Staubli VAL3: sendCommand.pgx

program sendCommand(num x_nCamID (dimensions=1), string x_sCmd (dimensions=1), bool& x_bError[] (dimensions=1))
  local string l_sMsgError
  local bool l_bError
  local num l_nErrorCode
begin
  //-----------------------------------------------------------------------
  //Header begin
  //Description of program
  //  Send native command to camera and read command execution error.
  //
  //Input parameters
  //  num x_nCamID :
  //    role : camera's ID
  //  string x_sCmd :
  //    role : native command
  //
  //Output parameters
  //  bool x_bError :
  //    role : returns true if operation suceeded and false otherwise
  //
  //Examples
  //  call sendCommand(l_nCamID,"tf"+x_sJob,l_bError)
  //
  //History
  //  Creation : 19-05-08 - f.Rob
  //Header end
  //-----------------------------------------------------------------------

  call writeSocket(x_nCamID,x_sCmd)
  call readSocket(x_nCamID,l_sMsgError,x_bError)
  call checkErrFormat(x_nCamID,l_sMsgError,l_bError)
  x_bError=l_bError
  if bDebugProgram
    //Displays error message
    //getFullError() replace getErrorCode() and getErrorMessage()
    call getFullError(x_nCamID,l_nErrorCode,l_sMsgError)
    ? "Cmd> "+l_sMsgError
  endIf
end
